FUNCTION_BLOCK FB_ComplexSheetStackerControl
VAR_INPUT

    //==============================================================
    // Group command inputs
    //==============================================================
    startCmd                            : BOOL;
    stopCmd                             : BOOL;
    resetCmd                            : BOOL;


    //==============================================================
    // Speed reference inputs
    //==============================================================
    lineSpeedMPM                        : REAL;

    // EN: Current sheet length [mm].
    // PT: Comprimento atual da chapa [mm].
    sheetLengthMm                       : REAL;


    //==============================================================
    // Package command input
    //==============================================================
    // EN: Rising edge starts package separation cycle.
    // PT: Borda de subida inicia o ciclo de separação do pacote.
    packageCompleteCmd                  : BOOL;
	sheetConveyorsSpeedUpCmd : BOOL;

    //==============================================================
    // Machine configuration
    //==============================================================
    machineConfig                       : ComplexStackerConfig_TypeStruct;


    //==============================================================
    // Safety input
    //==============================================================
    safetyCircuitOk                     : BOOL;


    //==============================================================
    // Synchronized conveyor drive status inputs
    //==============================================================
    sheetConveyor1DriveOk               : BOOL;
    sheetConveyor2DriveOk               : BOOL;
    sheetConveyor3DriveOk               : BOOL;
    sheetConveyor4DriveOk               : BOOL;
    elevatorDriveOk              : BOOL;


    //==============================================================
    // Auxiliary drive status inputs
    //==============================================================
    backstopDriveOk                     : BOOL;

	//==============================================================
	// Sheet stack discharge conveyor drive status input
	//==============================================================
    sheetStackDischargeConveyorDriveOk                 : BOOL;

	//==============================================================
	// EN: Stack buffer conveyor drive status inputs
	// PT: Entradas de estado dos acionamentos das esteiras buffer
	//==============================================================
	stackBufferConveyor1DriveOk            : BOOL;
	stackBufferConveyor2DriveOk            : BOOL;
	stackBufferConveyor3DriveOk            : BOOL;

	//==============================================================
	// EN: Stack detection sensors
	// PT: Sensores de detecção das pilhas
	//==============================================================
	stackBufferConveyor1StackPresentSensor : BOOL;
	stackBufferConveyor2StackPresentSensor : BOOL;
	stackBufferConveyor3StackPresentSensor : BOOL;
	elevatorStackPresentSensor             : BOOL;
	elevatorStackExitClearSensor           : BOOL;
	backstopMaterialInterlockSensor         : BOOL;
	backstopStackLevelSensor                : BOOL;

	
    //==============================================================
    // Position / measurement inputs
    //==============================================================
    stackHeightMm                       : REAL;
    backstopPositionMm                  : REAL;
    elevatorPositionMm           : REAL;


	//==============================================================
	// Elevator command inputs
	//==============================================================
	// EN: Starts elevator homing cycle.
	// PT: Inicia o ciclo de homing do elevador.
	elevatorHomeCmd              : BOOL;
	
	// EN: Enables elevator automatic mode. Auto-home is requested on
	//     startCmd and automatic leveling uses the stack level sensor.
	// PT: Habilita o modo automático do elevador. O auto-home é solicitado
	//     no startCmd e o nivelamento automático usa o sensor de nível da pilha.
	elevatorAutoCmd              : BOOL;
	
	// EN: Jog-up command in manual mode or during automatic leveling.
	// PT: Comando de jog para subir no manual ou durante o nivelamento automático.
	elevatorUpCmd                : BOOL;
	
	// EN: Jog-down command in manual mode or during automatic leveling.
	// PT: Comando de jog para descer no manual ou durante o nivelamento automático.
	elevatorDownCmd              : BOOL;


    //==============================================================
    // Elevator limit inputs
    //==============================================================
    elevatorUpperSafetyLimit     : BOOL;
    elevatorLowerSafetyLimit     : BOOL;

    elevatorUpperLimit           : BOOL;
    elevatorLowerLimit           : BOOL;


    //==============================================================
    // Backstop command inputs
    //==============================================================
    // EN: Starts the backstop homing cycle.
    // PT: Inicia o ciclo de homing do backstop.
    backstopHomeCmd                     : BOOL;
	
    // EN: Starts the backstop homing cycle.
    // PT: Inicia o ciclo de homing do backstop.
    backstopExecutePositioningCmd			 : BOOL;
    // EN: Enables automatic positioning according to sheet length.
    // PT: Habilita posicionamento automático conforme comprimento da chapa.
    backstopAutoCmd                     : BOOL;

    // EN: Manual open command.
    // PT: Comando manual para abrir.
    backstopOpenCmd                     : BOOL;

    // EN: Manual close command.
    // PT: Comando manual para fechar.
    backstopCloseCmd                    : BOOL;


    //==============================================================
    // Backstop limit inputs
    //==============================================================
    backstopSafeMaxLimit                    : BOOL;	
    backstopMaxLimit                 	   	: BOOL;
    backstopMinLimit                   		: BOOL;
    backstopSafeMinLimit                    : BOOL;


    //==============================================================
    // Sheet handling command inputs
    //==============================================================
	sheetStackDischargeConveyorManualRunCmd : BOOL;
    noCrushRollersDownCmd                 	: BOOL;

	// EN: Runs all three stack buffer conveyors.
	// PT: Aciona as três esteiras buffer de pilhas.
	stackBufferConveyorsRunCmd               : BOOL;

END_VAR


VAR_OUTPUT

	hmiAlarms : hmiAlarmsComplexStacker_TypeStruct;
	hmiStatus : hmiStatusComplexStacker_TypeStruct;
	stackerRunning : BOOL;
	alarmActive	: BOOL;
	stopMachinePulse : BOOL;
	reset 	: BOOL;
    //==============================================================
    // Synchronized conveyor drive outputs
    //==============================================================
    sheetConveyor1Run                   : BOOL;
    sheetConveyor2Run                   : BOOL;
    sheetConveyor3Run                   : BOOL;
    sheetConveyor4Run                   : BOOL;
	
	//==============================================================
	// Elevator drive outputs
	//==============================================================
	// EN: Elevator up run command.
	// PT: Comando para subir o elevador.
	elevatorRunUp                : BOOL;
	
	// EN: Elevator down run command.
	// PT: Comando para descer o elevador.
	elevatorRunDown              : BOOL;
	
	//==============================================================
	// Elevator magnetic brake output
	//==============================================================
	// EN: Magnetic brake release output. TRUE = brake released.
	// PT: Saída de liberação do freio magnético. TRUE = freio liberado.
	elevatorBrakeRelease         : BOOL;	

	// EN: Enables the elevator servo together with the stacker control.
	//     The servo remains enabled while stopped with zero speed reference.
	// PT: Habilita o servo do elevador junto com o controle do stacker.
	//     O servo permanece habilitado quando parado com referência zero.
	elevatorDriveEnable          : BOOL;

    //==============================================================
    // Backstop drive outputs
    //==============================================================
    // EN: Backstop forward run command. Positive/opening direction.
    // PT: Comando frente do backstop. Direção positiva/abrir.
    backstopRunFw                       : BOOL;

    // EN: Backstop reverse run command. Negative/closing direction.
    // PT: Comando reverso do backstop. Direção negativa/fechar.
    backstopRunRev                      : BOOL;

    // EN: Enables the backstop servo together with the stacker control.
    // PT: Habilita o servo do backstop junto com o controle do stacker.
    backstopDriveEnable                 : BOOL;

	//==============================================================
	// Sheet stack discharge conveyor outputs
	//==============================================================
	// EN: Sheet stack discharge conveyor run command.
	// PT: Comando de giro da esteira de descarga da pilha.
	sheetStackDischargeConveyorRun          : BOOL;

	//==============================================================
	// EN: Stack buffer conveyor run outputs
	// PT: Saídas de acionamento das esteiras buffer de pilhas
	//==============================================================
	stackBufferConveyor1Run                 : BOOL;
	stackBufferConveyor2Run                 : BOOL;
	stackBufferConveyor3Run                 : BOOL;




    //==============================================================
    // Synchronized conveyor speed reference outputs
    //==============================================================
    sheetConveyor1SpeedRefMPM           : REAL;
    sheetConveyor2SpeedRefMPM           : REAL;
    sheetConveyor3SpeedRefMPM           : REAL;
    sheetConveyor4SpeedRefMPM           : REAL;

    // EN: Signed elevator speed reference [mm/s]. Positive moves up
    //     and negative moves down.
    // PT: Referência de velocidade com sinal do elevador [mm/s].
    //     Positivo sobe e negativo desce.
    elevatorSpeedRefMmps                 : REAL;
	// EN: Sheet stack discharge conveyor speed reference [m/min].
	// PT: Referência de velocidade da esteira de descarga da pilha [m/min].
	sheetStackDischargeConveyorSpeedRefMPM  : REAL;

	// EN: Stack buffer conveyor speed references [m/min].
	// PT: Referências de velocidade das esteiras buffer [m/min].
	stackBufferConveyor1SpeedRefMPM         : REAL;
	stackBufferConveyor2SpeedRefMPM         : REAL;
	stackBufferConveyor3SpeedRefMPM         : REAL;

	// EN: TRUE while all three stack buffer positions are occupied.
	// PT: TRUE enquanto as três posições buffer estiverem ocupadas.
	stackBufferFull                         : BOOL;

	// EN: Requests the parent controller to reduce the machine speed.
	// PT: Solicita ao controlador pai a redução da velocidade da máquina.
	lineSpeedReductionRequest               : BOOL;

    //==============================================================
    // Backstop speed reference output
    //==============================================================
    // EN: Signed backstop speed reference [mm/s]. Positive opens and negative closes.
    // PT: Referência de velocidade com sinal do backstop [mm/s]. Positivo abre e negativo fecha.
    backstopSpeedRefMmps                : REAL;
	
	
	
    backstopPlateUpSolenoid                : BOOL;


    //==============================================================
    // Backstop encoder set outputs
    //==============================================================
    // EN: Pulse output to set/reset backstop encoder position.
    // PT: Pulso de saída para setar/resetar a posição do encoder do backstop.
    backstopSetEncoderPosition          : BOOL;

    // EN: Position value to set in the encoder block [mm].
    // PT: Valor de posição a ser gravado no bloco do encoder [mm].
    backstopSetEncoderPositionMm        : REAL;


    //==============================================================
    // Pneumatic valve outputs
    //==============================================================
    brakeValve                          : BOOL;

    sheetBrush1Valve                    : BOOL;
    sheetBrush2Valve                    : BOOL;
    sheetBrush3Valve                    : BOOL;

    brakeBrushValve                     : BOOL;
    backstopUpValve                     : BOOL;
    noCrushRollersUpDownValve               : BOOL;


    //==============================================================
    // General status outputs
    //==============================================================
    deviceState                         : STRING(30);

    faultActive                         : BOOL;
    synchronizedConveyorsRunning        : BOOL;


    //==============================================================
    // Sheet stack separation status outputs
    //==============================================================
    sheetStackSeparationState           : STRING(30);
    sheetStackSeparationStateCode       : INT;

    sheetStackSeparationReady           : BOOL;
    sheetStackSeparationActive          : BOOL;

    // EN: One-scan pulse when sheet stack separation starts.
    // PT: Pulso de um ciclo quando inicia a separação da pilha de chapas.
    sheetStackSeparationStarted         : BOOL;

    // EN: One-scan pulse when sheet stack separation finishes.
    // PT: Pulso de um ciclo quando finaliza a separação da pilha de chapas.
    sheetStackSeparationFinished        : BOOL;

    // EN: Brake active during sheet stack separation.
    // PT: Freio ativo durante a separação da pilha de chapas.
    sheetStackBrakeActive               : BOOL;


    //==============================================================
    // Sheet conveyor 2 separation status outputs
    //==============================================================
    sheetConveyor2SeparationActive      : BOOL;

    // EN: One-scan pulse when conveyor 2 separation tracking starts.
    // PT: Pulso de um ciclo quando inicia o rastreamento de separação da esteira 2.
    sheetConveyor2SeparationStarted     : BOOL;

    // EN: One-scan pulse when conveyor 2 separation tracking finishes.
    // PT: Pulso de um ciclo quando finaliza o rastreamento de separação da esteira 2.
    sheetConveyor2SeparationFinished    : BOOL;

    sheetConveyor2HighSpeedActive       : BOOL;

    // EN: Current conveyor 2 separation tracking distance [m].
    // PT: Distância atual rastreada na separação da esteira 2 [m].
    sheetConveyor2TrackingDistanceM     : REAL;

    // EN: Conveyor 2 separation target distance [m].
    // PT: Distância alvo de separação da esteira 2 [m].
    sheetConveyor2TargetDistanceM       : REAL;


    //==============================================================
    // Sheet conveyor 3 separation status outputs
    //==============================================================
    sheetConveyor3SeparationActive      : BOOL;

    // EN: One-scan pulse when conveyor 3 separation tracking starts.
    // PT: Pulso de um ciclo quando inicia o rastreamento de separação da esteira 3.
    sheetConveyor3SeparationStarted     : BOOL;

    // EN: One-scan pulse when conveyor 3 separation tracking finishes.
    // PT: Pulso de um ciclo quando finaliza o rastreamento de separação da esteira 3.
    sheetConveyor3SeparationFinished    : BOOL;

    sheetConveyor3HighSpeedActive       : BOOL;

    // EN: Current conveyor 3 separation tracking distance [m].
    // PT: Distância atual rastreada na separação da esteira 3 [m].
    sheetConveyor3TrackingDistanceM     : REAL;

    // EN: Conveyor 3 separation target distance [m].
    // PT: Distância alvo de separação da esteira 3 [m].
    sheetConveyor3TargetDistanceM       : REAL;

    //==============================================================
    // Sheet conveyor 4 separation status outputs
    //==============================================================
    sheetConveyor4SeparationActive      : BOOL;
    sheetConveyor4SeparationStarted     : BOOL;
    sheetConveyor4SeparationFinished    : BOOL;
    sheetConveyor4HighSpeedActive       : BOOL;
    sheetConveyor4TrackingDistanceM     : REAL;
    sheetConveyor4TargetDistanceM       : REAL;

	//==============================================================
	// Elevator encoder set outputs
	//==============================================================
	// EN: Pulse output to set/reset elevator encoder position.
	// PT: Pulso de saída para setar/resetar a posição do encoder do elevador.
	elevatorSetEncoderPosition   : BOOL;
	
	// EN: Position value to set in the elevator encoder block [mm].
	// PT: Valor de posição a ser gravado no bloco do encoder do elevador [mm].
	elevatorSetEncoderPositionMm : REAL;
	
	
	//==============================================================
	// Elevator status outputs
	//==============================================================
	elevatorState                : STRING(30);
	
	elevatorHomed                : BOOL;
	elevatorInPosition           : BOOL;

	// EN: TRUE when the homed elevator is at or below the configured
	//     minimum position considering the position tolerance.
	// PT: TRUE quando o elevador referenciado está na posição mínima
	//     configurada ou abaixo dela, considerando a tolerância.
	elevatorAtMinPosition        : BOOL;

	// EN: TRUE when the homed elevator is at or above the configured
	//     maximum position considering the position tolerance.
	// PT: TRUE quando o elevador referenciado está na posição máxima
	//     configurada ou acima dela, considerando a tolerância.
	elevatorAtMaxPosition        : BOOL;

	// EN: TRUE while manual jog speed is reduced near the endpoint
	//     toward which the elevator is moving.
	// PT: TRUE enquanto a velocidade do jog manual estiver reduzida próximo
	//     da extremidade para a qual o elevador está se movimentando.
	elevatorManualLowSpeedZoneActive : BOOL;

	elevatorFault                : BOOL;
	elevatorFaultCode            : INT;
	
	// EN: Current calculated elevator target position [mm].
	// PT: Posição alvo calculada atual do elevador [mm].
	elevatorTargetPositionMm     : REAL;
	
	// EN: Current elevator position error [mm].
	// PT: Erro atual de posição do elevador [mm].
	elevatorPositionErrorMm      : REAL;

    //==============================================================
    // Backstop status outputs
    //==============================================================
    backstopState                       : STRING(30);

    backstopHomed                       : BOOL;
    backstopInPosition                  : BOOL;
    backstopFault                       : BOOL;
    backstopFaultCode                   : INT;

    // EN: Current calculated target position [mm].
    // PT: Posição alvo calculada atualmente [mm].
    backstopTargetPositionMm            : REAL;

    // EN: Current position error [mm].
    // PT: Erro atual de posição [mm].
    backstopPositionErrorMm             : REAL;
	
	//==============================================================
	// Sheet stack discharge conveyor control state
	//==============================================================
	sheetStackDischargeConveyorState               : STRING(30);
	sheetStackDischargeConveyorFault               : BOOL;
	sheetStackDischargeConveyorFaultCode           : INT;
	
	//==============================================================
	// Sheet stack discharge sequence status outputs
	//==============================================================
	sheetStackDischargeState                : STRING(30);
	sheetStackDischargeStateCode            : INT;
	
	sheetStackDischargePending              : BOOL;
	sheetStackDischargeActive               : BOOL;
	sheetStackDischargeStarted              : BOOL;
	sheetStackDischargeFinished             : BOOL;
	
	sheetStackDischargeFault                : BOOL;
	sheetStackDischargeFaultCode            : INT;
	
	//==============================================================
	// Sheet stack discharge last cycle diagnostic outputs
	//==============================================================
	sheetStackDischargeLastCycleOk          : BOOL;
	sheetStackDischargeLastResultCode       : INT;
	sheetStackDischargeLastFaultStepCode    : INT;
	sheetStackDischargeLastFaultCode        : INT;	

END_VAR

VAR
	
	//==============================================================
	// Stop machine pulse control
	//==============================================================
	stopMachineFaultCondition     : BOOL;
	stopMachineFaultConditionOld  : BOOL;
	rStopMachineFaultCondition    : BOOL;
	
	tpStopMachinePulse            : TP;
	
	//==============================================================
	// Backstop manual intervention memory
	//==============================================================
	backstopManualInterventionActive     : BOOL;
	backstopManualInterventionPositionMm : REAL;
	
	//==============================================================
	// Sheet stack discharge backstop latched targets
	//==============================================================
	backstopProgrammedDischargeTargetMm : REAL;
	backstopDischargeOpenBasePositionMm : REAL;
	backstopDischargeOpenTargetMm       : REAL;
	
	//==============================================================
	// Backstop automatic positioning command control
	//==============================================================
	backstopExecutePositioningCmdOld    : BOOL;
	rBackstopExecutePositioning         : BOOL;
	
	backstopTargetOverrideOld           : BOOL;
	backstopTargetOverrideFallingEdge   : BOOL;
	
	backstopPositioningRequestActive    : BOOL;
	backstopLatchedTargetPositionMm     : REAL;
	backstopProgrammedTargetPositionMm  : REAL;
	
	//==============================================================
	// Backstop manual intervention memory
	//==============================================================
	// EN: Used by automatic discharge sequence to avoid closing onto material
	//     after operator manual intervention.

	//==============================================================
	// Backstop encoder set pulse
	//==============================================================
	backstopSetEncoderPositionTrigger  : BOOL;
	tpBackstopSetEncoderPosition       : TP;

	//==============================================================
	// Sheet stack discharge backstop latched targets
	//==============================================================

    //==============================================================
    // Group state machine
    //==============================================================
    syncConveyorsState                  : INT;


    //==============================================================
    // Package separation state machine
    //==============================================================
    packageSeparationState              : INT;


    //==============================================================
    // Backstop state machine
    //==============================================================
    backstopControlState                : INT;


    //==============================================================
    // Edge detection
    //==============================================================
    startCmdOld                         : BOOL;
    stopCmdOld                          : BOOL;
    packageCompleteCmdOld               : BOOL;

    backstopHomeCmdOld                  : BOOL;


    //==============================================================
    // Internal conditions
    //==============================================================
    allSynchronizedDrivesOk             : BOOL;
    anyFault                            : BOOL;
    speedControlEnabled                 : BOOL;
    rampReset                           : BOOL;


    //==============================================================
    // Sheet length conversion
    //==============================================================
    // EN: Internal sheet length converted from mm to m.
    // PT: Comprimento interno da chapa convertido de mm para m.
    sheetLengthM                        : REAL;


    //==============================================================
    // Normal speed calculation
    //==============================================================
    normalStackerSpeedMPM               : REAL;

    sheetConveyor1NormalSpeedMPM        : REAL;
    sheetConveyor2NormalSpeedMPM        : REAL;
    sheetConveyor3NormalSpeedMPM        : REAL;
    sheetConveyor4NormalSpeedMPM        : REAL;
    elevatorNormalSpeedMPM       : REAL;


    //==============================================================
    // Package gap speed calculation
    //==============================================================
    sheetConveyor2GapSpeedMPM           : REAL;
    sheetConveyor3GapSpeedMPM           : REAL;
    sheetConveyor4GapSpeedMPM           : REAL;


    //==============================================================
    // Speed targets
    //==============================================================
    sheetConveyor1TargetSpeedMPM        : REAL;
    sheetConveyor2TargetSpeedMPM        : REAL;
    sheetConveyor3TargetSpeedMPM        : REAL;
    sheetConveyor4TargetSpeedMPM        : REAL;
    elevatorTargetSpeedMPM       : REAL;


    //==============================================================
    // Package gap distance calculation
    //==============================================================
    packageGapDistanceTargetM           : REAL;

    sheetConveyor2OpeningSpeedMPM       : REAL;
    sheetConveyor3OpeningSpeedMPM       : REAL;
    sheetConveyor4OpeningSpeedMPM       : REAL;

    sheetConveyor2OpeningDistanceM      : REAL;
    sheetConveyor3OpeningDistanceM      : REAL;
    sheetConveyor4OpeningDistanceM      : REAL;


	//==============================================================
	// Elevator state machine
	//==============================================================
	elevatorControlState         : INT;
	
	
	//==============================================================
	// Elevator edge detection
	//==============================================================
	elevatorHomeCmdOld           : BOOL;
	rElevatorHome                : BOOL;
	
	
	//==============================================================
	// Elevator encoder set pulse
	//==============================================================
	elevatorSetEncoderPositionTrigger   : BOOL;
	tpElevatorSetEncoderPosition        : TP;
	
	
	//==============================================================
	// Elevator control calculation
	//==============================================================
	elevatorAutoTargetPositionMm        : REAL;
	elevatorRawSpeedRefMmps             : REAL;
	
	// EN: Internal signed speed command. Positive = up, negative = down.
	// PT: Comando interno de velocidade com sinal. Positivo = subir, negativo = descer.
	elevatorSignedSpeedRefMmps          : REAL;
	
	elevatorAbsPositionErrorMm          : REAL;
	
	
	//==============================================================
	// Elevator movement permissions
	//==============================================================
	elevatorUpAllowed                   : BOOL;
	elevatorDownAllowed                 : BOOL;
	
	elevatorMoveRequest                 : BOOL;
	elevatorBrakeReleaseRequest         : BOOL;
	
	
	//==============================================================
	// Elevator homing
	//==============================================================
	elevatorHomeLimitReached            : BOOL;
	elevatorHomeDownAllowed             : BOOL;
	elevatorHomeReleaseAllowed          : BOOL;
	elevatorManualCommandArmed          : BOOL;
	elevatorManualCommandRequest        : BOOL;
	elevatorReadyForAutomaticCycle      : BOOL;
	
	
	//==============================================================
	// Elevator timers
	//==============================================================
	tonElevatorHomingTimeout            : TON;
	tonElevatorHomeSettleDelay          : TON;
	tonElevatorLevelingSpeed2Delay      : TON;
	
	// EN: Delay after brake release before motor movement.
	// PT: Atraso após liberar o freio antes de movimentar o motor.
	tonElevatorBrakeReleaseDelay        : TON;
	
	// EN: Keeps brake released for a short time after movement stops.
	// PT: Mantém o freio liberado por um tempo após parar o movimento.
	tonElevatorBrakeHoldDelay           : TON;
	
	
	//==============================================================
	// Elevator speed ramp instance
	//==============================================================
	// EN: Ramp used for elevator vertical speed [mm/s].
	// PT: Rampa usada para velocidade vertical do elevador [mm/s].
	instRampElevator                    : FB_Gen_SRamp;
	

    //==============================================================
    // Backstop control calculation
    //==============================================================
    backstopAutoTargetPositionMm        : REAL;
    backstopRawSpeedRefMmps             : REAL;
    backstopAbsPositionErrorMm          : REAL;

    backstopHomeLimitReached            : BOOL;
    backstopOpenAllowed                 : BOOL;
    backstopCloseAllowed                : BOOL;

    rBackstopHome                       : BOOL;


	//==============================================================
	// Backstop homing edge detection
	//==============================================================
	backstopHomeLimitOld                 : BOOL;
	backstopHomeLimitFallingEdge         : BOOL;
	backstopHomeMoveAllowed              : BOOL;
	
	
	
	//==============================================================
	// Backstop timers
	//==============================================================
	tonBackstopHomeSettleDelay           : TON;



    //==============================================================
    // Backstop timers
    //==============================================================
    tonBackstopHomingTimeout            : TON;


    //==============================================================
    // Speed ramp instances
    //==============================================================
    instRampSheetConveyor1              : FB_Gen_SRamp;
    instRampSheetConveyor2              : FB_Gen_SRamp;
    instRampSheetConveyor3              : FB_Gen_SRamp;
    instRampSheetConveyor4              : FB_Gen_SRamp;


    //==============================================================
    // PLC scan time measurement
    //==============================================================
    instCycleTime                       : CYCLE_TIME;
    scanTimeS                           : REAL;
    scanTimeMs                          : REAL;

	backstopSignedSpeedRefMmps: REAL;
	
	//==============================================================
	// Sheet stack discharge state machine
	//==============================================================
	sheetStackDischargeControlState         : INT;
	
	
	//==============================================================
	// Sheet stack discharge edge detection
	//==============================================================
	packageCompleteCmdOldDischarge          : BOOL;
	rPackageCompleteDischarge               : BOOL;
	
	
	//==============================================================
	// Sheet stack discharge timers
	//==============================================================
	tonSheetStackDischarge                  : TON;
	tonSheetStackDischargePlatformClearTimeout : TON;
	elevatorPlatformClearDetected           : BOOL;
	elevatorStackPresentAtDischargeStart    : BOOL;
	
	
	//==============================================================
	// Sheet stack discharge internal conditions
	//==============================================================
	sheetStackDischargeFaultCondition       : BOOL;
	
	
	//==============================================================
	// Backstop target override
	//==============================================================
	backstopTargetOverrideActive            : BOOL;
	backstopTargetOverridePositionMm        : REAL;
	backstopRequiredForAutomaticOperation   : BOOL;
	
	
	//==============================================================
	// Elevator target override
	//==============================================================
	elevatorTargetOverrideActive     : BOOL;
	elevatorTargetOverridePositionMm : REAL;	
	
	
	sheetStackDischargeConveyorRunRequest: BOOL;
	instTONBackstopDownDelay: TON;
	
	//==============================================================
	// Sheet stack discharge step timeout
	//==============================================================
	tonSheetStackDischargeStepTimeout       : TON;
	
	sheetStackDischargeCycleHasManualSkip   : BOOL;
	sheetStackDischargeCycleHasTimeout      : BOOL;	
	
	
	//==============================================================
	// Elevator homing edge detection
	//==============================================================
	elevatorHomeLimitOld                 : BOOL;
	elevatorHomeLimitFallingEdge         : BOOL;	

	//==============================================================
	// System master run control
	//==============================================================
	systemRunEnable : BOOL;
	
	rStartCmd : BOOL;
	rStopCmd  : BOOL;
	
	//==============================================================
	// Automatic homing requests generated by master start
	//==============================================================
	backstopAutoHomeRequest        : BOOL;
	elevatorAutoHomeRequest : BOOL;
	
	//==============================================================
	// Elevator home request command control
	//==============================================================
	elevatorHomeRequestCombined    : BOOL;
	elevatorHomeRequestCombinedOld : BOOL;
	backstopHomeRunning: BOOL;
	//==============================================================
	// Backstop home request command control
	//==============================================================
	backstopHomeRequestCombined    : BOOL;
	backstopHomeRequestCombinedOld : BOOL;

	//==============================================================
	// EN: Stack buffer conveyor control
	// PT: Controle das esteiras buffer de pilhas
	//==============================================================
	stackBufferControlState                 : INT;
	stackBufferTargetConveyor               : INT;
	elevatorStackExitClearSensorOld         : BOOL;
	rElevatorStackExitClear                 : BOOL;
	tonStackBufferStopDelay                 : TON;
	tonStackBufferTransferTimeout           : TON;
	tonStackBufferFullSpeedReduction        : TON;
	
END_VAR

_SystemControl();

_SheetConveyorGroupControl();
_ConveyorSpeedControl();

_SheetStackDischargeControl();

_BackstopControl();
_ElevatorControl();
_SheetStackDischargeConveyorControl();
_StackBufferConveyorsControl();
_MachineAuxilary();
_HmiStatus();
_AlarmControl();

//==============================================================
// COMPLEX STACKER — ALARM CONTROL
// EN: Maps internal faults and status conditions to HMI alarm structure.
//==============================================================
METHOD _AlarmControl

VAR
	hmiAlarmsNotActive: hmiAlarmsComplexStacker_TypeStruct;
END_VAR
//==============================================================
// HMI alarms reset / latch logic
//==============================================================

IF resetCmd THEN

    // Reset geral dos alarmes
    hmiAlarms := hmiAlarmsNotActive;

ELSE

    //==============================================================
    // 1) General / system alarms
    //==============================================================
    hmiAlarms.safetyCircuitNotOk :=
        hmiAlarms.safetyCircuitNotOk OR
        NOT safetyCircuitOk;

    hmiAlarms.systemFaultActive :=
        hmiAlarms.systemFaultActive OR
        faultActive OR
        (
            backstopRequiredForAutomaticOperation AND
            backstopFault
        ) OR
        elevatorFault OR
        sheetStackDischargeFault OR
        sheetStackDischargeConveyorFault OR
        NOT stackBufferConveyor1DriveOk OR
        NOT stackBufferConveyor2DriveOk OR
        NOT stackBufferConveyor3DriveOk;

    hmiAlarms.systemNotEnabled :=
        hmiAlarms.systemNotEnabled OR
        NOT systemRunEnable;


    //==============================================================
    // 2) Sheet conveyor group alarms
    //==============================================================
    hmiAlarms.sheetConveyor1DriveNotOk :=
        hmiAlarms.sheetConveyor1DriveNotOk OR
        NOT sheetConveyor1DriveOk;

    hmiAlarms.sheetConveyor2DriveNotOk :=
        hmiAlarms.sheetConveyor2DriveNotOk OR
        NOT sheetConveyor2DriveOk;

    hmiAlarms.sheetConveyor3DriveNotOk :=
        hmiAlarms.sheetConveyor3DriveNotOk OR
        NOT sheetConveyor3DriveOk;

    hmiAlarms.sheetConveyor4DriveNotOk :=
        hmiAlarms.sheetConveyor4DriveNotOk OR
        NOT sheetConveyor4DriveOk;

    hmiAlarms.sheetConveyorGroupFault :=
        hmiAlarms.sheetConveyorGroupFault OR
        NOT safetyCircuitOk OR
        NOT sheetConveyor1DriveOk OR
        NOT sheetConveyor2DriveOk OR
        NOT sheetConveyor3DriveOk OR
        NOT sheetConveyor4DriveOk;


    //==============================================================
    // 2.1) Stack buffer conveyor alarms
    // EN: Buffer drive faults are alarmed without stopping the main
    //     synchronized conveyor group automatically.
    // PT: Falhas dos drives do buffer geram alarme sem parar automaticamente
    //     o grupo principal de esteiras sincronizadas.
    //==============================================================
    hmiAlarms.stackBufferConveyor1DriveNotOk :=
        hmiAlarms.stackBufferConveyor1DriveNotOk OR
        NOT stackBufferConveyor1DriveOk;

    hmiAlarms.stackBufferConveyor2DriveNotOk :=
        hmiAlarms.stackBufferConveyor2DriveNotOk OR
        NOT stackBufferConveyor2DriveOk;

    hmiAlarms.stackBufferConveyor3DriveNotOk :=
        hmiAlarms.stackBufferConveyor3DriveNotOk OR
        NOT stackBufferConveyor3DriveOk;

    hmiAlarms.stackBufferConveyorGroupFault :=
        hmiAlarms.stackBufferConveyorGroupFault OR
        NOT safetyCircuitOk OR
        NOT stackBufferConveyor1DriveOk OR
        NOT stackBufferConveyor2DriveOk OR
        NOT stackBufferConveyor3DriveOk;

 //   hmiAlarms.synchronizedConveyorsNotRunning :=
 //       hmiAlarms.synchronizedConveyorsNotRunning OR
 //       (
 //           systemRunEnable AND
 //           NOT synchronizedConveyorsRunning
 //       );


    //==============================================================
    // 3) Sheet stack separation alarms / indications
    //==============================================================
    // Mantido comentado conforme lógica original.
    // Se quiser ativar como latch, use o mesmo padrão:
    //
    // hmiAlarms.sheetStackSeparationNotReady :=
    //     hmiAlarms.sheetStackSeparationNotReady OR
    //     (
    //         systemRunEnable AND
    //         synchronizedConveyorsRunning AND
    //         NOT sheetStackSeparationReady
    //     );
    //
    // hmiAlarms.sheetStackSeparationActive :=
    //     hmiAlarms.sheetStackSeparationActive OR
    //     sheetStackSeparationActive;
    //
    // hmiAlarms.sheetStackBrakeActive :=
    //     hmiAlarms.sheetStackBrakeActive OR
    //     sheetStackBrakeActive;


    //==============================================================
    // 4) Sheet stack discharge sequence alarms / indications
    //==============================================================
    hmiAlarms.sheetStackDischargeFault :=
        hmiAlarms.sheetStackDischargeFault OR
        sheetStackDischargeFault;

    hmiAlarms.sheetStackDischargeLastCycleNotOk :=
        hmiAlarms.sheetStackDischargeLastCycleNotOk OR
        (
            NOT sheetStackDischargeLastCycleOk AND
            sheetStackDischargeLastResultCode <> 0
        );

    hmiAlarms.sheetStackDischargeTimeout :=
        hmiAlarms.sheetStackDischargeTimeout OR
        sheetStackDischargeLastResultCode = 3;

    hmiAlarms.sheetStackDischargeManualSkip :=
        hmiAlarms.sheetStackDischargeManualSkip OR
        sheetStackDischargeLastResultCode = 2;


    //==============================================================
    // 5) Sheet stack discharge conveyor alarms
    //==============================================================
    hmiAlarms.sheetStackDischargeConveyorDriveNotOk :=
        hmiAlarms.sheetStackDischargeConveyorDriveNotOk OR
        NOT sheetStackDischargeConveyorDriveOk;

    hmiAlarms.sheetStackDischargeConveyorFault :=
        hmiAlarms.sheetStackDischargeConveyorFault OR
        sheetStackDischargeConveyorFault;


    //==============================================================
    // 6) Backstop alarms / indications
    //==============================================================
    hmiAlarms.backstopDriveNotOk :=
        hmiAlarms.backstopDriveNotOk OR
        NOT backstopDriveOk;

    hmiAlarms.backstopFault :=
        hmiAlarms.backstopFault OR
        backstopFault;

    hmiAlarms.backstopNotHomed :=
        hmiAlarms.backstopNotHomed OR
        (
            backstopAutoCmd AND
            NOT backstopHomed
        );

    (*
    hmiAlarms.backstopNotInPosition :=
        hmiAlarms.backstopNotInPosition OR
        (
            systemRunEnable AND
            backstopAutoCmd AND
            backstopHomed AND
            NOT backstopInPosition AND
            NOT backstopTargetOverrideActive
        );
    *)

    hmiAlarms.backstopSafeMaxLimitActive :=
        hmiAlarms.backstopSafeMaxLimitActive OR
        backstopSafeMaxLimit;

    hmiAlarms.backstopSafeMinLimitActive :=
        hmiAlarms.backstopSafeMinLimitActive OR
        backstopSafeMinLimit;

    (*
    hmiAlarms.backstopMaxLimitActive :=
        hmiAlarms.backstopMaxLimitActive OR
        backstopMaxLimit;

    hmiAlarms.backstopMinLimitActive :=
        hmiAlarms.backstopMinLimitActive OR
        backstopMinLimit;

    hmiAlarms.backstopManualInterventionActive :=
        hmiAlarms.backstopManualInterventionActive OR
        backstopManualInterventionActive;
    *)


    //==============================================================
    // 7) Elevator alarms / indications
    //==============================================================
    hmiAlarms.elevatorDriveNotOk :=
        hmiAlarms.elevatorDriveNotOk OR
        NOT elevatorDriveOk;

    hmiAlarms.elevatorFault :=
        hmiAlarms.elevatorFault OR
        elevatorFault;

    hmiAlarms.elevatorNotHomed :=
        hmiAlarms.elevatorNotHomed OR
        (
            elevatorAutoCmd AND
            NOT elevatorHomed
        );

//    hmiAlarms.elevatorNotInPosition :=
//        hmiAlarms.elevatorNotInPosition OR
//        (
//            systemRunEnable AND
//            elevatorAutoCmd AND
//            elevatorHomed AND
//            NOT elevatorInPosition
//        );

    hmiAlarms.elevatorUpperSafetyLimitActive :=
        hmiAlarms.elevatorUpperSafetyLimitActive OR
        elevatorUpperSafetyLimit;

    hmiAlarms.elevatorLowerSafetyLimitActive :=
        hmiAlarms.elevatorLowerSafetyLimitActive OR
        elevatorLowerSafetyLimit;

    (*
    hmiAlarms.elevatorUpperLimitActive :=
        hmiAlarms.elevatorUpperLimitActive OR
        elevatorUpperLimit;

    hmiAlarms.elevatorLowerLimitActive :=
        hmiAlarms.elevatorLowerLimitActive OR
        elevatorLowerLimit;
    *)

END_IF;
END_METHOD

//==============================================================
// COMPLEX STACKER — BACKSTOP CONTROL
// EN: Controls the backstop axis with homing, manual movement,
//     automatic positioning, override positioning and protections.
//
// Signed speed convention:
// Positive = open
// Negative = close
//
// State code:
// 0  = STOP
// 10 = HOME_FAST_SEARCH
// 11 = HOME_SLOW_EXIT_SENSOR
// 12 = HOME_SET_ENCODER
// 13 = HOME_WAIT_AFTER_SET
// 14 = HOME_MOVE_TO_TARGET
// 20 = MANUAL
// 30 = AUTO_POSITION
// 40 = FAULT
//==============================================================
METHOD _BackstopControl



//==============================================================
// 1) Default internal commands
//==============================================================
// EN: Internal signed speed is reset every scan and set by the active state.
//     Positive = open, negative = close.
backstopSignedSpeedRefMmps := 0.0;

// EN: Internal trigger for encoder set pulse.
backstopSetEncoderPositionTrigger := FALSE;


//==============================================================
// 2) Edge detection
//==============================================================
// EN: Home can be requested manually by HMI or automatically by _SystemControl.
//     Automatic home is accepted only when backstopAutoCmd is enabled.
//     Movement is allowed only when master system run is enabled.
backstopHomeRequestCombined :=
    systemRunEnable AND
    (
        backstopHomeCmd OR
        (
            backstopAutoCmd AND
            backstopAutoHomeRequest
        )
    );

rBackstopHome :=
    backstopHomeRequestCombined AND
    NOT backstopHomeRequestCombinedOld;

backstopHomeRequestCombinedOld :=
    backstopHomeRequestCombined;


// EN: Execute positioning command edge.
//     This command only generates movement when system is enabled and backstop auto is enabled.
rBackstopExecutePositioning :=
    systemRunEnable AND
    backstopExecutePositioningCmd AND
    NOT backstopExecutePositioningCmdOld;

backstopExecutePositioningCmdOld := backstopExecutePositioningCmd;


// EN: Override falling edge.
//     Used as fallback to return to programmed position if override is released.
backstopTargetOverrideFallingEdge :=
    backstopTargetOverrideOld AND NOT backstopTargetOverrideActive;

backstopTargetOverrideOld := backstopTargetOverrideActive;


//==============================================================
// 3) Home limit selection and edge detection
//==============================================================
// EN: Home limit depends on configured homing direction.
IF machineConfig.backstopHomeDirection > 0 THEN

    backstopHomeLimitReached := backstopMaxLimit;

ELSIF machineConfig.backstopHomeDirection < 0 THEN

    backstopHomeLimitReached := backstopMinLimit;

ELSE

    backstopHomeLimitReached := FALSE;

END_IF;


// EN: Falling edge is used after the home limit has been reached.
backstopHomeLimitFallingEdge :=
    backstopHomeLimitOld AND NOT backstopHomeLimitReached;

backstopHomeLimitOld := backstopHomeLimitReached;


//==============================================================
// 4) Movement permissions
//==============================================================
backstopOpenAllowed :=
    systemRunEnable AND
    safetyCircuitOk AND
    backstopDriveOk AND
    NOT backstopMaxLimit AND
    NOT backstopSafeMaxLimit AND
    (
        (NOT backstopHomed) OR
        (backstopPositionMm < machineConfig.backstopMaxPositionMm)
    );

backstopCloseAllowed :=
    systemRunEnable AND
    safetyCircuitOk AND
    backstopDriveOk AND
    NOT backstopMinLimit AND
    NOT backstopSafeMinLimit AND
    (
        (NOT backstopHomed) OR
        (backstopPositionMm > machineConfig.backstopMinPositionMm)
    );


// EN: During homing, the normal home limit is allowed.
//     Only the safe limit blocks movement.
IF machineConfig.backstopHomeDirection > 0 THEN

    backstopHomeMoveAllowed :=
        systemRunEnable AND
        safetyCircuitOk AND
        backstopDriveOk AND
        NOT backstopSafeMaxLimit;

ELSIF machineConfig.backstopHomeDirection < 0 THEN

    backstopHomeMoveAllowed :=
        systemRunEnable AND
        safetyCircuitOk AND
        backstopDriveOk AND
        NOT backstopSafeMinLimit;

ELSE

    backstopHomeMoveAllowed := FALSE;

END_IF;


//==============================================================
// 5) Programmed / override target calculation
//==============================================================
// EN: Programmed target follows sheet length plus mechanical offset.
//     This value can change, but it does not move the backstop by itself.
backstopProgrammedTargetPositionMm :=
    LIMIT(
        machineConfig.backstopMinPositionMm,
        MAX(0.0, sheetLengthMm) + machineConfig.backstopSheetLengthOffsetMm,
        machineConfig.backstopMaxPositionMm
    );


// EN: Before homing, keep the latched target updated with programmed target.
//     This avoids an invalid old target after power-up.
IF NOT backstopHomed THEN

    backstopLatchedTargetPositionMm := backstopProgrammedTargetPositionMm;

END_IF;


//==============================================================
// 5.1) Automatic positioning request handling
//==============================================================
// EN: Auto mode only enables positioning. It does not execute positioning.
//     Normal positioning must be requested by backstopExecutePositioningCmd.
//     Override positioning is requested by the automatic cycle.
IF NOT systemRunEnable THEN

    backstopPositioningRequestActive := FALSE;


ELSIF NOT backstopAutoCmd THEN

    backstopPositioningRequestActive := FALSE;


ELSIF backstopTargetOverrideActive THEN

    // EN: Override has priority. Clear normal positioning request.
    backstopPositioningRequestActive := FALSE;


ELSIF rBackstopExecutePositioning THEN

    // EN: Latch current programmed target only when execute command is received.
    backstopLatchedTargetPositionMm := backstopProgrammedTargetPositionMm;
    backstopPositioningRequestActive := TRUE;


ELSIF backstopTargetOverrideFallingEdge THEN

    // EN: Fallback after override release.
    //     The discharge sequence should normally keep override active
    //     during return. If override is released unexpectedly, return to
    //     programmed position automatically.
    backstopLatchedTargetPositionMm := backstopProgrammedTargetPositionMm;
    backstopPositioningRequestActive := TRUE;

END_IF;


//==============================================================
// 5.2) Active target selection
//==============================================================
// EN: Discharge override is accepted only while the backstop is in automatic.
//     In manual mode the backstop is completely independent from the cycle.
// PT: O override de descarte é aceito somente com o backstop em automático.
//     No modo manual o backstop fica completamente independente do ciclo.
IF systemRunEnable AND
   backstopAutoCmd AND
   backstopTargetOverrideActive THEN

    backstopTargetPositionMm :=
        LIMIT(
            machineConfig.backstopMinPositionMm,
            backstopTargetOverridePositionMm,
            machineConfig.backstopMaxPositionMm
        );

ELSE

    backstopTargetPositionMm :=
        LIMIT(
            machineConfig.backstopMinPositionMm,
            backstopLatchedTargetPositionMm,
            machineConfig.backstopMaxPositionMm
        );

END_IF;


//==============================================================
// 5.4) Home running flag
//==============================================================
IF (backstopControlState = 10) OR
   (backstopControlState = 11) OR
   (backstopControlState = 12) OR
   (backstopControlState = 13) OR
   (backstopControlState = 14) THEN

    backstopHomeRunning := TRUE;

ELSE

    backstopHomeRunning := FALSE;

END_IF;


//==============================================================
// 6) Position error calculation
//==============================================================
backstopPositionErrorMm :=
    backstopTargetPositionMm - backstopPositionMm;

backstopAbsPositionErrorMm :=
    ABS(backstopPositionErrorMm);

backstopInPosition :=
    backstopHomed AND
    (backstopAbsPositionErrorMm <= machineConfig.backstopPositionToleranceMm);


//==============================================================
// 7) Reset fault command
//==============================================================
IF resetCmd THEN

    IF safetyCircuitOk AND
       backstopDriveOk AND
       NOT backstopSafeMaxLimit AND
       NOT backstopSafeMinLimit THEN

        backstopFault := FALSE;
        backstopFaultCode := 0;

        IF backstopControlState = 40 THEN
            backstopControlState := 0;
        END_IF

    END_IF

END_IF;


//==============================================================
// 8) General protection
//==============================================================
IF NOT safetyCircuitOk THEN

    backstopState := 'SAFETY_OFF';

    tonBackstopHomingTimeout(IN := FALSE);
    tonBackstopHomeSettleDelay(IN := FALSE);

    backstopFault := TRUE;
    backstopFaultCode := 2;
    backstopControlState := 40;


ELSIF NOT backstopDriveOk THEN

    backstopState := 'DRIVE_NOT_OK';

    tonBackstopHomingTimeout(IN := FALSE);
    tonBackstopHomeSettleDelay(IN := FALSE);

    backstopFault := TRUE;
    backstopFaultCode := 1;
    backstopControlState := 40;


ELSIF backstopSafeMaxLimit THEN

    backstopState := 'SAFE_MAX_LIMIT';

    tonBackstopHomingTimeout(IN := FALSE);
    tonBackstopHomeSettleDelay(IN := FALSE);

    backstopFault := TRUE;
    backstopFaultCode := 6;
    backstopControlState := 40;


ELSIF backstopSafeMinLimit THEN

    backstopState := 'SAFE_MIN_LIMIT';

    tonBackstopHomingTimeout(IN := FALSE);
    tonBackstopHomeSettleDelay(IN := FALSE);

    backstopFault := TRUE;
    backstopFaultCode := 7;
    backstopControlState := 40;


ELSIF machineConfig.backstopHomeDirection = 0 THEN

    backstopState := 'INVALID_HOME_DIR';

    tonBackstopHomingTimeout(IN := FALSE);
    tonBackstopHomeSettleDelay(IN := FALSE);

    backstopFault := TRUE;
    backstopFaultCode := 5;
    backstopControlState := 40;


ELSIF NOT systemRunEnable THEN

    // EN: Master stop disables movement without generating an axis fault.
    backstopState := 'SYSTEM_DISABLED';

    backstopSignedSpeedRefMmps := 0.0;

    tonBackstopHomingTimeout(IN := FALSE);
    tonBackstopHomeSettleDelay(IN := FALSE);

    backstopPositioningRequestActive := FALSE;

    IF backstopControlState <> 40 THEN
        backstopControlState := 0;
    END_IF


ELSE

    //==============================================================
    // 9) Mode selection
    //==============================================================
    // EN: Homing has priority over manual and automatic positioning.
    IF rBackstopHome AND NOT backstopFault THEN
        backstopControlState := 10;
    END_IF;


    //==============================================================
    // 10) Backstop state machine
    //==============================================================
    CASE backstopControlState OF

        0: // STOP
            backstopState := 'STOP';

            tonBackstopHomingTimeout(IN := FALSE);
            tonBackstopHomeSettleDelay(IN := FALSE);

            // EN: Manual is allowed even with auto enabled,
            //     but not during an automatic cycle override.
            IF (backstopOpenCmd OR backstopCloseCmd) AND
               NOT (
                   backstopAutoCmd AND
                   backstopTargetOverrideActive
               ) THEN

                backstopControlState := 20;


            ELSIF backstopAutoCmd AND
                  (
                      backstopTargetOverrideActive OR
                      backstopPositioningRequestActive
                  ) THEN

                backstopControlState := 30;

            END_IF


        10: // HOME_FAST_SEARCH
            backstopState := 'HOME_FAST';

            backstopHomed := FALSE;
            backstopInPosition := FALSE;

            tonBackstopHomeSettleDelay(IN := FALSE);

            tonBackstopHomingTimeout(
                IN := TRUE,
                PT := machineConfig.backstopHomingTimeout
            );

            IF tonBackstopHomingTimeout.Q THEN

                backstopSignedSpeedRefMmps := 0.0;

                tonBackstopHomingTimeout(IN := FALSE);

                backstopFault := TRUE;
                backstopFaultCode := 3;

                backstopState := 'HOME_TIMEOUT';
                backstopControlState := 40;


            ELSIF backstopHomeLimitReached THEN

                backstopSignedSpeedRefMmps := 0.0;

                backstopControlState := 11;


            ELSE

                IF backstopHomeMoveAllowed THEN

                    IF machineConfig.backstopHomeDirection > 0 THEN

                        backstopSignedSpeedRefMmps :=
                            ABS(machineConfig.backstopHomingSpeedMmps);

                    ELSE

                        backstopSignedSpeedRefMmps :=
                            -ABS(machineConfig.backstopHomingSpeedMmps);

                    END_IF

                ELSE

                    backstopSignedSpeedRefMmps := 0.0;

                END_IF

            END_IF


        11: // HOME_SLOW_EXIT_SENSOR
            backstopState := 'HOME_SLOW_EXIT';

            tonBackstopHomeSettleDelay(IN := FALSE);

            tonBackstopHomingTimeout(
                IN := TRUE,
                PT := machineConfig.backstopHomingTimeout
            );

            IF tonBackstopHomingTimeout.Q THEN

                backstopSignedSpeedRefMmps := 0.0;

                tonBackstopHomingTimeout(IN := FALSE);

                backstopFault := TRUE;
                backstopFaultCode := 3;

                backstopState := 'HOME_TIMEOUT';
                backstopControlState := 40;


            ELSIF backstopHomeLimitFallingEdge THEN

                backstopSignedSpeedRefMmps := 0.0;

                tonBackstopHomingTimeout(IN := FALSE);

                backstopControlState := 12;


            ELSE

                IF backstopHomeMoveAllowed THEN

                    IF machineConfig.backstopHomeDirection > 0 THEN

                        backstopSignedSpeedRefMmps :=
                            -ABS(machineConfig.backstopMinMoveSpeedMmps);

                    ELSE

                        backstopSignedSpeedRefMmps :=
                            ABS(machineConfig.backstopMinMoveSpeedMmps);

                    END_IF

                ELSE

                    backstopSignedSpeedRefMmps := 0.0;

                END_IF

            END_IF


        12: // HOME_SET_ENCODER
            backstopState := 'HOME_SET_ENCODER';

            backstopSignedSpeedRefMmps := 0.0;

            tonBackstopHomingTimeout(IN := FALSE);
            tonBackstopHomeSettleDelay(IN := FALSE);

            // EN: Set encoder to configured known home position.
            backstopSetEncoderPositionTrigger := TRUE;
            backstopSetEncoderPositionMm := machineConfig.backstopHomePositionMm;

            backstopHomed := TRUE;
            backstopFault := FALSE;
            backstopFaultCode := 0;

            // EN: After homing, latch current programmed target for home move.
            backstopLatchedTargetPositionMm := backstopProgrammedTargetPositionMm;
            backstopPositioningRequestActive := TRUE;

            // EN: Homing cancels previous manual intervention memory.
            backstopManualInterventionActive := FALSE;
            backstopManualInterventionPositionMm := 0.0;

            backstopControlState := 13;


        13: // HOME_WAIT_AFTER_SET
            backstopState := 'HOME_WAIT';

            backstopSignedSpeedRefMmps := 0.0;

            tonBackstopHomingTimeout(IN := FALSE);

            // EN: Fixed wait after encoder set.
            tonBackstopHomeSettleDelay(
                IN := TRUE,
                PT := T#5S
            );

            IF tonBackstopHomeSettleDelay.Q THEN

                tonBackstopHomeSettleDelay(IN := FALSE);

                backstopControlState := 14;

            END_IF


        14: // HOME_MOVE_TO_TARGET
            backstopState := 'HOME_TO_TARGET';

            tonBackstopHomingTimeout(IN := FALSE);
            tonBackstopHomeSettleDelay(IN := FALSE);

            // EN: Move to the latched programmed target after homing.
            IF backstopInPosition THEN

                backstopSignedSpeedRefMmps := 0.0;

                backstopPositioningRequestActive := FALSE;

                // EN: Home positioning completed, no manual intervention pending.
                backstopManualInterventionActive := FALSE;
                backstopManualInterventionPositionMm := 0.0;

                backstopControlState := 0;


            ELSE

                backstopRawSpeedRefMmps :=
                    backstopPositionErrorMm * machineConfig.backstopPositionKp;

                backstopRawSpeedRefMmps :=
                    LIMIT(
                        -ABS(machineConfig.backstopAutoMaxSpeedMmps),
                        backstopRawSpeedRefMmps,
                        ABS(machineConfig.backstopAutoMaxSpeedMmps)
                    );

                IF ABS(backstopRawSpeedRefMmps) <
                   ABS(machineConfig.backstopMinMoveSpeedMmps) THEN

                    IF backstopPositionErrorMm > 0.0 THEN

                        backstopRawSpeedRefMmps :=
                            ABS(machineConfig.backstopMinMoveSpeedMmps);

                    ELSE

                        backstopRawSpeedRefMmps :=
                            -ABS(machineConfig.backstopMinMoveSpeedMmps);

                    END_IF

                END_IF

                IF (backstopRawSpeedRefMmps > 0.0) AND backstopOpenAllowed THEN

                    backstopSignedSpeedRefMmps := backstopRawSpeedRefMmps;

                ELSIF (backstopRawSpeedRefMmps < 0.0) AND backstopCloseAllowed THEN

                    backstopSignedSpeedRefMmps := backstopRawSpeedRefMmps;

                ELSE

                    backstopSignedSpeedRefMmps := 0.0;

                END_IF

            END_IF


        20: // MANUAL
            backstopState := 'MANUAL';

            tonBackstopHomingTimeout(IN := FALSE);
            tonBackstopHomeSettleDelay(IN := FALSE);

            // EN: An automatic override cancels manual control only when
            //     the backstop itself is enabled in automatic mode.
            // PT: O override automático cancela o controle manual somente
            //     quando o próprio backstop está habilitado em automático.
            IF backstopAutoCmd AND
               backstopTargetOverrideActive THEN

                backstopSignedSpeedRefMmps := 0.0;
                backstopControlState := 30;


            ELSIF backstopOpenCmd AND backstopCloseCmd THEN

                backstopSignedSpeedRefMmps := 0.0;


            ELSIF backstopOpenCmd THEN

                IF backstopOpenAllowed THEN

                    backstopSignedSpeedRefMmps :=
                        ABS(machineConfig.backstopManualSpeedMmps);

                    // EN: Store last manual intervention position.
                    //     This is updated while the operator holds the manual command.
                    backstopManualInterventionActive := TRUE;
                    backstopManualInterventionPositionMm := backstopPositionMm;

                ELSE

                    backstopSignedSpeedRefMmps := 0.0;

                END_IF


            ELSIF backstopCloseCmd THEN

                IF backstopCloseAllowed THEN

                    backstopSignedSpeedRefMmps :=
                        -ABS(machineConfig.backstopManualSpeedMmps);

                    // EN: Store last manual intervention position.
                    //     Even if operator closes, the discharge sequence will use
                    //     MAX(programmed position, manual position), so it remains safe.
                    backstopManualInterventionActive := TRUE;
                    backstopManualInterventionPositionMm := backstopPositionMm;

                ELSE

                    backstopSignedSpeedRefMmps := 0.0;

                END_IF


            ELSE

                backstopSignedSpeedRefMmps := 0.0;

                // EN: After manual command release, do not automatically return
                //     to programmed position. Wait for execute positioning command.
                backstopPositioningRequestActive := FALSE;

                backstopControlState := 0;

            END_IF


        30: // AUTO_POSITION
            backstopState := 'AUTO_POSITION';

            tonBackstopHomingTimeout(IN := FALSE);
            tonBackstopHomeSettleDelay(IN := FALSE);

            // EN: Manual mode always cancels automatic positioning,
            //     regardless of any external override request.
            // PT: O modo manual sempre cancela o posicionamento automático,
            //     independentemente de qualquer pedido externo de override.
            IF NOT backstopAutoCmd THEN

                backstopSignedSpeedRefMmps := 0.0;
                backstopPositioningRequestActive := FALSE;
                backstopControlState := 0;


            ELSIF NOT backstopHomed THEN

                backstopSignedSpeedRefMmps := 0.0;
                backstopState := 'AUTO_NO_HOME';


            ELSIF (backstopOpenCmd OR backstopCloseCmd) AND
                  NOT backstopTargetOverrideActive THEN

                // EN: Manual has priority only outside automatic cycle override.
                backstopSignedSpeedRefMmps := 0.0;
                backstopPositioningRequestActive := FALSE;
                backstopControlState := 20;


            ELSIF NOT backstopTargetOverrideActive AND
                  NOT backstopPositioningRequestActive THEN

                // EN: Auto enabled but no positioning command active.
                backstopSignedSpeedRefMmps := 0.0;
                backstopControlState := 0;


            ELSIF backstopInPosition THEN

                backstopSignedSpeedRefMmps := 0.0;

                // EN: Normal positioning command ends when target is reached.
                //     Override remains controlled by the automatic cycle.
                IF NOT backstopTargetOverrideActive THEN

                    backstopPositioningRequestActive := FALSE;

                    // EN: If the backstop returned to programmed target,
                    //     clear previous manual intervention memory.
                    backstopManualInterventionActive := FALSE;
                    backstopManualInterventionPositionMm := 0.0;

                    backstopControlState := 0;

                END_IF


            ELSE

                backstopRawSpeedRefMmps :=
                    backstopPositionErrorMm * machineConfig.backstopPositionKp;

                backstopRawSpeedRefMmps :=
                    LIMIT(
                        -ABS(machineConfig.backstopAutoMaxSpeedMmps),
                        backstopRawSpeedRefMmps,
                        ABS(machineConfig.backstopAutoMaxSpeedMmps)
                    );

                IF ABS(backstopRawSpeedRefMmps) <
                   ABS(machineConfig.backstopMinMoveSpeedMmps) THEN

                    IF backstopPositionErrorMm > 0.0 THEN

                        backstopRawSpeedRefMmps :=
                            ABS(machineConfig.backstopMinMoveSpeedMmps);

                    ELSE

                        backstopRawSpeedRefMmps :=
                            -ABS(machineConfig.backstopMinMoveSpeedMmps);

                    END_IF

                END_IF

                IF (backstopRawSpeedRefMmps > 0.0) AND backstopOpenAllowed THEN

                    backstopSignedSpeedRefMmps := backstopRawSpeedRefMmps;

                ELSIF (backstopRawSpeedRefMmps < 0.0) AND backstopCloseAllowed THEN

                    backstopSignedSpeedRefMmps := backstopRawSpeedRefMmps;

                ELSE

                    backstopSignedSpeedRefMmps := 0.0;

                END_IF

            END_IF


        40: // FAULT
            backstopState := 'FAULT';

            backstopSignedSpeedRefMmps := 0.0;

            tonBackstopHomingTimeout(IN := FALSE);
            tonBackstopHomeSettleDelay(IN := FALSE);

            backstopPositioningRequestActive := FALSE;

            IF resetCmd AND
               safetyCircuitOk AND
               backstopDriveOk AND
               NOT backstopSafeMaxLimit AND
               NOT backstopSafeMinLimit THEN

                backstopFault := FALSE;
                backstopFaultCode := 0;
                backstopControlState := 0;

            END_IF


    ELSE

        backstopControlState := 0;

    END_CASE;

END_IF;


//==============================================================
// 11) Encoder set pulse
//==============================================================
// EN: Extend encoder set command to ensure the encoder block sees it.
tpBackstopSetEncoderPosition(
    IN := backstopSetEncoderPositionTrigger,
    PT := machineConfig.backstopSetEncoderPulseTime
);

backstopSetEncoderPosition := tpBackstopSetEncoderPosition.Q;


//==============================================================
// 12) Backstop drive direction and speed outputs
//==============================================================
// EN: Convert signed internal speed command into direction outputs
//     and positive speed reference.
IF systemRunEnable AND
   safetyCircuitOk AND
   backstopDriveOk AND
   NOT backstopFault AND
   (ABS(backstopSignedSpeedRefMmps) >= machineConfig.backstopRunMinSpeedMmps) THEN

    // EN: The servo receives the signed speed reference directly.
    // PT: O servo recebe diretamente a referência de velocidade com sinal.
    backstopSpeedRefMmps := backstopSignedSpeedRefMmps;

    backstopRunFw :=
        backstopSignedSpeedRefMmps > 0.0;

    backstopRunRev :=
        backstopSignedSpeedRefMmps < 0.0;

ELSE

    backstopSpeedRefMmps := 0.0;

    backstopRunFw := FALSE;
    backstopRunRev := FALSE;

END_IF;

// EN: Enable the servo with the stacker system; drive-ready feedback is not used here
//     because it would create a circular enable dependency.
// PT: Habilita o servo com o sistema do stacker; o retorno de drive pronto não é usado
//     aqui porque criaria uma dependência circular de habilitação.
backstopDriveEnable := systemRunEnable AND safetyCircuitOk;


//==============================================================
// 13) Backstop plate lift solenoid
//==============================================================
// EN: Lift the backstop plate during backstop movement and homing.
//     Discharge conveyor protection can be ORed after all methods are called.
IF systemRunEnable AND
   (
       backstopRunFw OR
       backstopRunRev OR
       sheetStackDischargeConveyorRun OR
       (backstopControlState = 10) OR
       (backstopControlState = 11) OR
       (backstopControlState = 12) OR
       (backstopControlState = 13) OR
       (backstopControlState = 14)
   ) THEN

    backstopPlateUpSolenoid := TRUE;
    instTONBackstopDownDelay.IN := FALSE;

ELSE

    instTONBackstopDownDelay.IN := TRUE;

    IF instTONBackstopDownDelay.Q THEN

        backstopPlateUpSolenoid := FALSE;

    END_IF

END_IF;

instTONBackstopDownDelay(PT := T#200MS);
END_METHOD

//==============================================================
// COMPLEX STACKER — SPEED REFERENCE GENERATOR
// EN: Generates synchronized and sheet-stack separation speed references [m/min].
//==============================================================
METHOD _ConveyorSpeedControl
VAR
    rPackageComplete                  : BOOL;
    packageGapReady                   : BOOL;
    validCycleTimeS                   : REAL;

    sheetConveyorsSpeedUpReferenceMPM : REAL;

    sheetConveyor1BaseSpeedMPM        : REAL;
    sheetConveyor2BaseSpeedMPM        : REAL;
    sheetConveyor3BaseSpeedMPM        : REAL;
    sheetConveyor4BaseSpeedMPM        : REAL;
END_VAR


//==============================================================
// 1) Default event pulses
//==============================================================
sheetStackSeparationStarted         := FALSE;
sheetStackSeparationFinished        := FALSE;

sheetConveyor2SeparationStarted     := FALSE;
sheetConveyor2SeparationFinished    := FALSE;

sheetConveyor3SeparationStarted     := FALSE;
sheetConveyor3SeparationFinished    := FALSE;

sheetConveyor4SeparationStarted     := FALSE;
sheetConveyor4SeparationFinished    := FALSE;


//==============================================================
// 2) Edge detection
//==============================================================
rPackageComplete := packageCompleteCmd AND NOT packageCompleteCmdOld;
packageCompleteCmdOld := packageCompleteCmd;


//==============================================================
// 3) Enable and scan time
//==============================================================
speedControlEnabled :=
    sheetConveyor1Run AND
    sheetConveyor2Run AND
    sheetConveyor3Run AND
    sheetConveyor4Run AND
    safetyCircuitOk;

rampReset := NOT speedControlEnabled;


// EN: Read PLC scan time using OSCAT CYCLE_TIME.
instCycleTime(
    RST := resetCmd
);


// EN: Convert last cycle time from TIME/ms to seconds.
scanTimeMs := TIME_TO_REAL(instCycleTime.ct_last);

validCycleTimeS :=
    LIMIT(
        0.001,
        scanTimeMs / 1000.0,
        20.0
    );

scanTimeS := validCycleTimeS;


//==============================================================
// 4) Sheet length conversion
//==============================================================
// EN: Sheet length is kept converted for other calculations,
//     but it is no longer used as the separation tracking target.
sheetLengthM := MAX(0.0, sheetLengthMm) / 1000.0;


//==============================================================
// 5) Calculate normal stacker speed
//==============================================================
IF speedControlEnabled THEN

    normalStackerSpeedMPM :=
        LIMIT(
            machineConfig.minimumSpeedMPM,
            MAX(0.0, lineSpeedMPM) *
                MAX(0.0, machineConfig.stackerSpeedRatio),
            machineConfig.maximumSpeedMPM
        );

ELSE

    normalStackerSpeedMPM := 0.0;

END_IF;


//==============================================================
// 6) Calculate normal speed for each conveyor
//==============================================================
sheetConveyor1NormalSpeedMPM :=
    normalStackerSpeedMPM *
    MAX(0.0, machineConfig.sheetConveyor1SpeedTrim);

sheetConveyor2NormalSpeedMPM :=
    normalStackerSpeedMPM *
    MAX(0.0, machineConfig.sheetConveyor2SpeedTrim);

sheetConveyor3NormalSpeedMPM :=
    normalStackerSpeedMPM *
    MAX(0.0, machineConfig.sheetConveyor3SpeedTrim);

sheetConveyor4NormalSpeedMPM :=
    normalStackerSpeedMPM *
    MAX(0.0, machineConfig.sheetConveyor4SpeedTrim);


//==============================================================
// 6.1) Sheet conveyors speed-up reference
//==============================================================
// EN: Speed-up is added directly to conveyors 1/2/3 references.
//     It can work even when line speed is zero, as long as the
//     conveyor group is enabled.
IF speedControlEnabled AND sheetConveyorsSpeedUpCmd THEN

    sheetConveyorsSpeedUpReferenceMPM :=
        MAX(0.0, machineConfig.sheetConveyorsSpeedUpMPM);

ELSE

    sheetConveyorsSpeedUpReferenceMPM := 0.0;

END_IF;


//==============================================================
// 6.2) Base speed references including speed-up
//==============================================================
// EN: Base speed is the synchronized conveyor speed plus operator speed-up.
//     Separation tracking must use this base speed as reference.
sheetConveyor1BaseSpeedMPM :=
    sheetConveyor1NormalSpeedMPM + sheetConveyorsSpeedUpReferenceMPM;

sheetConveyor2BaseSpeedMPM :=
    sheetConveyor2NormalSpeedMPM + sheetConveyorsSpeedUpReferenceMPM;

sheetConveyor3BaseSpeedMPM :=
    sheetConveyor3NormalSpeedMPM + sheetConveyorsSpeedUpReferenceMPM;

sheetConveyor4BaseSpeedMPM :=
    sheetConveyor4NormalSpeedMPM + sheetConveyorsSpeedUpReferenceMPM;


//==============================================================
// 7) Calculate separation high speed
//==============================================================
// EN: Gap speed also receives the same speed-up reference.
//     This preserves the real gap differential while allowing operator boost.
sheetConveyor2GapSpeedMPM :=
    (sheetConveyor2NormalSpeedMPM * MAX(0.0, machineConfig.packageGapSpeedRatio)) +
    machineConfig.packageGapSpeedOffsetMPM +
    sheetConveyorsSpeedUpReferenceMPM;

sheetConveyor3GapSpeedMPM :=
    (sheetConveyor3NormalSpeedMPM * MAX(0.0, machineConfig.packageGapSpeedRatio)) +
    machineConfig.packageGapSpeedOffsetMPM +
    sheetConveyorsSpeedUpReferenceMPM;

sheetConveyor4GapSpeedMPM :=
    (sheetConveyor4NormalSpeedMPM * MAX(0.0, machineConfig.packageGapSpeedRatio)) +
    machineConfig.packageGapSpeedOffsetMPM +
    sheetConveyorsSpeedUpReferenceMPM;


//==============================================================
// 8) Calculate separation tracking target distances
//==============================================================
// EN: Separation tracking target is based on each conveyor length.
sheetConveyor2TargetDistanceM :=
    MAX(0.0, machineConfig.sheetConveyor2LengthM);

sheetConveyor3TargetDistanceM :=
    MAX(0.0, machineConfig.sheetConveyor3LengthM);

sheetConveyor4TargetDistanceM :=
    MAX(0.0, machineConfig.sheetConveyor4LengthM);


//==============================================================
// 9) Check separation ready conditions
//==============================================================
// EN: Compare gap speed against base speed, not normal speed.
//     Otherwise operator speed-up would be incorrectly counted as gap opening.
packageGapReady :=
    speedControlEnabled AND
    (sheetConveyor2TargetDistanceM > 0.0) AND
    (sheetConveyor3TargetDistanceM > 0.0) AND
    (sheetConveyor4TargetDistanceM > 0.0) AND
    ((sheetConveyor2GapSpeedMPM - sheetConveyor2BaseSpeedMPM) >= machineConfig.minimumOpeningSpeedMPM) AND
    ((sheetConveyor3GapSpeedMPM - sheetConveyor3BaseSpeedMPM) >= machineConfig.minimumOpeningSpeedMPM) AND
    ((sheetConveyor4GapSpeedMPM - sheetConveyor4BaseSpeedMPM) >= machineConfig.minimumOpeningSpeedMPM);

sheetStackSeparationReady := packageGapReady;


//==============================================================
// 10) Sheet stack separation state machine
//==============================================================
IF NOT speedControlEnabled THEN

    sheetStackSeparationState      := 'DISABLED';
    sheetStackSeparationStateCode  := -1;

    packageSeparationState         := 0;

    sheetStackSeparationActive     := FALSE;
    sheetStackBrakeActive          := FALSE;
    brakeValve                     := FALSE;

    sheetConveyor2SeparationActive := FALSE;
    sheetConveyor3SeparationActive := FALSE;
    sheetConveyor4SeparationActive := FALSE;

    sheetConveyor2HighSpeedActive  := FALSE;
    sheetConveyor3HighSpeedActive  := FALSE;
    sheetConveyor4HighSpeedActive  := FALSE;

    sheetConveyor2OpeningDistanceM := 0.0;
    sheetConveyor3OpeningDistanceM := 0.0;
    sheetConveyor4OpeningDistanceM := 0.0;

    sheetConveyor1TargetSpeedMPM   := 0.0;
    sheetConveyor2TargetSpeedMPM   := 0.0;
    sheetConveyor3TargetSpeedMPM   := 0.0;
    sheetConveyor4TargetSpeedMPM   := 0.0;


ELSE

    CASE packageSeparationState OF

        0: // NORMAL
            sheetStackSeparationState     := 'NORMAL';
            sheetStackSeparationStateCode := 0;

            sheetStackSeparationActive    := FALSE;
            sheetStackBrakeActive         := FALSE;
            brakeValve                    := FALSE;

            sheetConveyor2SeparationActive := FALSE;
            sheetConveyor3SeparationActive := FALSE;
            sheetConveyor4SeparationActive := FALSE;

            sheetConveyor2HighSpeedActive  := FALSE;
            sheetConveyor3HighSpeedActive  := FALSE;
            sheetConveyor4HighSpeedActive  := FALSE;

            sheetConveyor2OpeningDistanceM := 0.0;
            sheetConveyor3OpeningDistanceM := 0.0;
            sheetConveyor4OpeningDistanceM := 0.0;

            sheetConveyor1TargetSpeedMPM  := sheetConveyor1BaseSpeedMPM;
            sheetConveyor2TargetSpeedMPM  := sheetConveyor2BaseSpeedMPM;
            sheetConveyor3TargetSpeedMPM  := sheetConveyor3BaseSpeedMPM;
            sheetConveyor4TargetSpeedMPM  := sheetConveyor4BaseSpeedMPM;

            IF rPackageComplete AND packageGapReady THEN
                packageSeparationState := 10;
            END_IF


        10: // START_SHEET_STACK_SEPARATION
            sheetStackSeparationState     := 'START_SEPARATION';
            sheetStackSeparationStateCode := 10;

            sheetStackSeparationActive    := TRUE;
            sheetStackSeparationStarted   := TRUE;

            sheetStackBrakeActive         := TRUE;
            brakeValve                    := TRUE;

            // EN: Conveyor 2 tracking starts immediately.
            sheetConveyor2SeparationStarted := TRUE;

            sheetConveyor2SeparationActive  := TRUE;
            sheetConveyor3SeparationActive  := FALSE;
            sheetConveyor4SeparationActive  := FALSE;

            // EN: Conveyor 2 and 3 accelerate together from the beginning.
            sheetConveyor2HighSpeedActive   := TRUE;
            sheetConveyor3HighSpeedActive   := TRUE;
            sheetConveyor4HighSpeedActive   := TRUE;

            sheetConveyor2OpeningDistanceM  := 0.0;
            sheetConveyor3OpeningDistanceM  := 0.0;
            sheetConveyor4OpeningDistanceM  := 0.0;

            sheetConveyor1TargetSpeedMPM    := sheetConveyor1BaseSpeedMPM;
            sheetConveyor2TargetSpeedMPM    := sheetConveyor2GapSpeedMPM;
            sheetConveyor3TargetSpeedMPM    := sheetConveyor3GapSpeedMPM;
            sheetConveyor4TargetSpeedMPM    := sheetConveyor4GapSpeedMPM;

            packageSeparationState := 20;


        20: // SHEET_CONVEYOR_2_SEPARATION_TRACKING
            sheetStackSeparationState     := 'CONV2_TRACKING';
            sheetStackSeparationStateCode := 20;

            sheetStackSeparationActive    := TRUE;

            sheetStackBrakeActive         := TRUE;
            brakeValve                    := TRUE;

            sheetConveyor2SeparationActive := TRUE;
            sheetConveyor3SeparationActive := FALSE;
            sheetConveyor4SeparationActive := FALSE;

            sheetConveyor2HighSpeedActive  := TRUE;
            sheetConveyor3HighSpeedActive  := TRUE;
            sheetConveyor4HighSpeedActive  := TRUE;

            sheetConveyor1TargetSpeedMPM  := sheetConveyor1BaseSpeedMPM;
            sheetConveyor2TargetSpeedMPM  := sheetConveyor2GapSpeedMPM;
            sheetConveyor3TargetSpeedMPM  := sheetConveyor3GapSpeedMPM;
            sheetConveyor4TargetSpeedMPM  := sheetConveyor4GapSpeedMPM;

            IF sheetConveyor2OpeningDistanceM >= sheetConveyor2TargetDistanceM THEN

                // EN: Conveyor 2 tracking finished. Conveyor 2 returns to base speed.
                sheetConveyor2SeparationFinished := TRUE;

                sheetConveyor2SeparationActive   := FALSE;
                sheetConveyor2HighSpeedActive    := FALSE;

                sheetStackBrakeActive            := FALSE;
                brakeValve                       := FALSE;

                sheetConveyor2TargetSpeedMPM     := sheetConveyor2BaseSpeedMPM;

                // EN: Conveyor 3 tracking starts after conveyor 2 returns to sync.
                sheetConveyor3SeparationStarted := TRUE;
                sheetConveyor3OpeningDistanceM  := 0.0;

                packageSeparationState := 30;

            END_IF


        30: // SHEET_CONVEYOR_3_SEPARATION_TRACKING
            sheetStackSeparationState     := 'CONV3_TRACKING';
            sheetStackSeparationStateCode := 30;

            sheetStackSeparationActive    := TRUE;

            sheetStackBrakeActive         := FALSE;
            brakeValve                    := FALSE;

            sheetConveyor2SeparationActive := FALSE;
            sheetConveyor3SeparationActive := TRUE;
            sheetConveyor4SeparationActive := FALSE;

            sheetConveyor2HighSpeedActive  := FALSE;
            sheetConveyor3HighSpeedActive  := TRUE;
            sheetConveyor4HighSpeedActive  := TRUE;

            sheetConveyor1TargetSpeedMPM  := sheetConveyor1BaseSpeedMPM;
            sheetConveyor2TargetSpeedMPM  := sheetConveyor2BaseSpeedMPM;
            sheetConveyor3TargetSpeedMPM  := sheetConveyor3GapSpeedMPM;
            sheetConveyor4TargetSpeedMPM  := sheetConveyor4GapSpeedMPM;

            IF sheetConveyor3OpeningDistanceM >= sheetConveyor3TargetDistanceM THEN

                // EN: Conveyor 3 returns to base synchronized speed.
                sheetConveyor3TargetSpeedMPM := sheetConveyor3BaseSpeedMPM;

                // EN: Conveyor 4 tracking starts after conveyor 3 returns to sync.
                // PT: O rastreamento da esteira 4 inicia após a esteira 3 retornar ao sincronismo.
                sheetConveyor4SeparationStarted := TRUE;
                sheetConveyor4OpeningDistanceM := 0.0;

                packageSeparationState := 40;

            END_IF


        40: // SHEET_CONVEYOR_4_SEPARATION_TRACKING
            sheetStackSeparationState     := 'CONV4_TRACKING';
            sheetStackSeparationStateCode := 40;

            sheetStackSeparationActive    := TRUE;
            sheetStackBrakeActive         := FALSE;
            brakeValve                    := FALSE;

            sheetConveyor2SeparationActive := FALSE;
            sheetConveyor3SeparationActive := FALSE;
            sheetConveyor4SeparationActive := TRUE;

            sheetConveyor2HighSpeedActive := FALSE;
            sheetConveyor3HighSpeedActive := FALSE;
            sheetConveyor4HighSpeedActive := TRUE;

            sheetConveyor1TargetSpeedMPM := sheetConveyor1BaseSpeedMPM;
            sheetConveyor2TargetSpeedMPM := sheetConveyor2BaseSpeedMPM;
            sheetConveyor3TargetSpeedMPM := sheetConveyor3BaseSpeedMPM;
            sheetConveyor4TargetSpeedMPM := sheetConveyor4GapSpeedMPM;

            IF sheetConveyor4OpeningDistanceM >= sheetConveyor4TargetDistanceM THEN
                sheetConveyor4TargetSpeedMPM := sheetConveyor4BaseSpeedMPM;
                packageSeparationState := 50;
            END_IF


        50: // FINISH_SHEET_STACK_SEPARATION
            sheetStackSeparationState     := 'FINISH_SEPARATION';
            sheetStackSeparationStateCode := 50;

            sheetStackSeparationActive    := FALSE;
            sheetStackSeparationFinished  := TRUE;

            sheetStackBrakeActive         := FALSE;
            brakeValve                    := FALSE;

            sheetConveyor2SeparationActive  := FALSE;
            sheetConveyor3SeparationActive  := FALSE;
            sheetConveyor4SeparationActive  := FALSE;

            sheetConveyor2HighSpeedActive   := FALSE;
            sheetConveyor3HighSpeedActive   := FALSE;
            sheetConveyor4HighSpeedActive   := FALSE;

            sheetConveyor3SeparationFinished := TRUE;
            sheetConveyor4SeparationFinished := TRUE;

            sheetConveyor1TargetSpeedMPM  := sheetConveyor1BaseSpeedMPM;
            sheetConveyor2TargetSpeedMPM  := sheetConveyor2BaseSpeedMPM;
            sheetConveyor3TargetSpeedMPM  := sheetConveyor3BaseSpeedMPM;
            sheetConveyor4TargetSpeedMPM  := sheetConveyor4BaseSpeedMPM;

            packageSeparationState := 0;


    ELSE

        packageSeparationState := 0;

    END_CASE;

END_IF;


//==============================================================
// 11) Limit speed targets
//==============================================================
sheetConveyor1TargetSpeedMPM := LIMIT(
    machineConfig.minimumSpeedMPM,
    sheetConveyor1TargetSpeedMPM,
    machineConfig.maximumSpeedMPM
);

sheetConveyor2TargetSpeedMPM := LIMIT(
    machineConfig.minimumSpeedMPM,
    sheetConveyor2TargetSpeedMPM,
    machineConfig.maximumSpeedMPM
);

sheetConveyor3TargetSpeedMPM := LIMIT(
    machineConfig.minimumSpeedMPM,
    sheetConveyor3TargetSpeedMPM,
    machineConfig.maximumSpeedMPM
);

sheetConveyor4TargetSpeedMPM := LIMIT(
    machineConfig.minimumSpeedMPM,
    sheetConveyor4TargetSpeedMPM,
    machineConfig.maximumSpeedMPM
);


//==============================================================
// 12) Ramp sheet conveyor 1 speed reference
//==============================================================
instRampSheetConveyor1(
    X          := sheetConveyor1TargetSpeedMPM,
    A_UP       := MAX(0.0, machineConfig.rampAccelerationUpMPMps2),
    A_DN       := -MAX(0.0, machineConfig.rampAccelerationDownMPMps2),
    VU_MAX     := MAX(0.0, machineConfig.rampVelocityUpMaxMPMps),
    VD_MAX     := -MAX(0.0, machineConfig.rampVelocityDownMaxMPMps),
    LIMIT_HIGH := machineConfig.maximumSpeedMPM,
    LIMIT_LOW  := machineConfig.minimumSpeedMPM,
    RST        := rampReset,
    Y          => sheetConveyor1SpeedRefMPM
);


//==============================================================
// 13) Ramp sheet conveyor 2 speed reference
//==============================================================
instRampSheetConveyor2(
    X          := sheetConveyor2TargetSpeedMPM,
    A_UP       := MAX(0.0, machineConfig.rampAccelerationUpMPMps2),
    A_DN       := -MAX(0.0, machineConfig.rampAccelerationDownMPMps2),
    VU_MAX     := MAX(0.0, machineConfig.rampVelocityUpMaxMPMps),
    VD_MAX     := -MAX(0.0, machineConfig.rampVelocityDownMaxMPMps),
    LIMIT_HIGH := machineConfig.maximumSpeedMPM,
    LIMIT_LOW  := machineConfig.minimumSpeedMPM,
    RST        := rampReset,
    Y          => sheetConveyor2SpeedRefMPM
);


//==============================================================
// 14) Ramp sheet conveyor 3 speed reference
//==============================================================
instRampSheetConveyor3(
    X          := sheetConveyor3TargetSpeedMPM,
    A_UP       := MAX(0.0, machineConfig.rampAccelerationUpMPMps2),
    A_DN       := -MAX(0.0, machineConfig.rampAccelerationDownMPMps2),
    VU_MAX     := MAX(0.0, machineConfig.rampVelocityUpMaxMPMps),
    VD_MAX     := -MAX(0.0, machineConfig.rampVelocityDownMaxMPMps),
    LIMIT_HIGH := machineConfig.maximumSpeedMPM,
    LIMIT_LOW  := machineConfig.minimumSpeedMPM,
    RST        := rampReset,
    Y          => sheetConveyor3SpeedRefMPM
);


//==============================================================
// 15) Ramp sheet conveyor 4 speed reference
//==============================================================
instRampSheetConveyor4(
    X          := sheetConveyor4TargetSpeedMPM,
    A_UP       := MAX(0.0, machineConfig.rampAccelerationUpMPMps2),
    A_DN       := -MAX(0.0, machineConfig.rampAccelerationDownMPMps2),
    VU_MAX     := MAX(0.0, machineConfig.rampVelocityUpMaxMPMps),
    VD_MAX     := -MAX(0.0, machineConfig.rampVelocityDownMaxMPMps),
    LIMIT_HIGH := machineConfig.maximumSpeedMPM,
    LIMIT_LOW  := machineConfig.minimumSpeedMPM,
    RST        := rampReset,
    Y          => sheetConveyor4SpeedRefMPM
);


//==============================================================
// 16) Calculate real separation tracking speed using ramped references
//==============================================================
// EN: Only the real speed differential above the base speed moves the
//     separation point through the conveyors.
//     Operator speed-up is already included in base speed, so it is not
//     counted as gap opening.
sheetConveyor2OpeningSpeedMPM :=
    MAX(0.0, sheetConveyor2SpeedRefMPM - sheetConveyor2BaseSpeedMPM);

sheetConveyor3OpeningSpeedMPM :=
    MAX(0.0, sheetConveyor3SpeedRefMPM - sheetConveyor3BaseSpeedMPM);

sheetConveyor4OpeningSpeedMPM :=
    MAX(0.0, sheetConveyor4SpeedRefMPM - sheetConveyor4BaseSpeedMPM);


//==============================================================
// 17) Integrate real separation tracking distance
//==============================================================
IF speedControlEnabled THEN

    IF packageSeparationState = 20 THEN

        IF sheetConveyor2OpeningSpeedMPM >= machineConfig.minimumOpeningSpeedMPM THEN

            sheetConveyor2OpeningDistanceM :=
                sheetConveyor2OpeningDistanceM +
                (sheetConveyor2OpeningSpeedMPM / 60.0) * scanTimeS;

        END_IF

    ELSIF packageSeparationState = 30 THEN

        IF sheetConveyor3OpeningSpeedMPM >= machineConfig.minimumOpeningSpeedMPM THEN

            sheetConveyor3OpeningDistanceM :=
                sheetConveyor3OpeningDistanceM +
                (sheetConveyor3OpeningSpeedMPM / 60.0) * scanTimeS;

        END_IF

    ELSIF packageSeparationState = 40 THEN

        IF sheetConveyor4OpeningSpeedMPM >= machineConfig.minimumOpeningSpeedMPM THEN

            sheetConveyor4OpeningDistanceM :=
                sheetConveyor4OpeningDistanceM +
                (sheetConveyor4OpeningSpeedMPM / 60.0) * scanTimeS;

        END_IF

    END_IF

END_IF;


//==============================================================
// 18) Publish tracking distances to outputs
//==============================================================
sheetConveyor2TrackingDistanceM := sheetConveyor2OpeningDistanceM;
sheetConveyor3TrackingDistanceM := sheetConveyor3OpeningDistanceM;
sheetConveyor4TrackingDistanceM := sheetConveyor4OpeningDistanceM;
END_METHOD

//==============================================================
// COMPLEX STACKER - ELEVATOR CONTROL
// EN: Controls homing, manual movement, automatic leveling,
//     discharge positioning and magnetic brake timing.
// PT: Controla homing, movimento manual, nivelamento automático,
//     posicionamento de descarga e temporização do freio magnético.
//
// Signed speed: positive = up; negative = down.
// Velocidade com sinal: positivo = subir; negativo = descer.
//
// State code:
// 0  = STOP
// 10 = HOME_DOWN_SEARCH
// 11 = HOME_RELEASE_SENSOR
// 12 = HOME_SETTLE
// 13 = HOME_SET_ENCODER
// 14 = HOME_MOVE_TO_UPPER_POSITION
// 20 = MANUAL
// 30 = AUTO_LEVELING
// 40 = DISCHARGE_POSITIONING
// 90 = FAULT
//==============================================================
METHOD _ElevatorControl
//==============================================================
// 1) Default internal commands
//==============================================================
elevatorSignedSpeedRefMmps := 0.0;
elevatorSetEncoderPositionTrigger := FALSE;
elevatorManualLowSpeedZoneActive := FALSE;


//==============================================================
// 2) Homing request and lower sensor edge detection
//==============================================================
elevatorHomeRequestCombined :=
    systemRunEnable AND
    (
        elevatorHomeCmd OR
        (
            elevatorAutoCmd AND
            elevatorAutoHomeRequest
        )
    );

rElevatorHome :=
    elevatorHomeRequestCombined AND
    NOT elevatorHomeRequestCombinedOld;

elevatorHomeRequestCombinedOld := elevatorHomeRequestCombined;

elevatorHomeLimitReached := elevatorLowerLimit;

elevatorHomeLimitFallingEdge :=
    elevatorHomeLimitOld AND
    NOT elevatorHomeLimitReached;

elevatorHomeLimitOld := elevatorHomeLimitReached;


//==============================================================
// 2.1) Manual command rearm
//==============================================================
// EN: Manual commands held during homing or active discharge positioning
//     must be released before a new manual movement can start.
//     Waiting for stack separation keeps leveling and manual control active.
// PT: Comandos manuais mantidos durante homing ou posicionamento ativo de
//     descarte devem ser liberados antes que um novo movimento manual inicie.
//     A espera pela separação mantém o nivelamento e o controle manual ativos.
IF NOT systemRunEnable OR
   NOT safetyCircuitOk OR
   NOT elevatorDriveOk OR
   elevatorFault OR
   (
        (elevatorControlState >= 10) AND
        (elevatorControlState <= 14)
   ) OR
   (elevatorControlState = 40) OR
   (elevatorControlState = 90) OR
   elevatorTargetOverrideActive OR
   sheetStackDischargeActive THEN

    elevatorManualCommandArmed := FALSE;

ELSIF NOT elevatorUpCmd AND
      NOT elevatorDownCmd THEN

    elevatorManualCommandArmed := TRUE;

END_IF;

elevatorManualCommandRequest :=
    elevatorManualCommandArmed AND
    (elevatorUpCmd OR elevatorDownCmd);


//==============================================================
// 3) Movement permissions
//==============================================================
elevatorUpAllowed :=
    systemRunEnable AND
    safetyCircuitOk AND
    elevatorDriveOk AND
    NOT elevatorUpperLimit AND
    NOT elevatorUpperSafetyLimit AND
    NOT backstopMaterialInterlockSensor AND
    (
        (NOT elevatorHomed) OR
        (elevatorPositionMm < machineConfig.elevatorMaxPositionMm)
    );

elevatorDownAllowed :=
    systemRunEnable AND
    safetyCircuitOk AND
    elevatorDriveOk AND
    NOT elevatorLowerLimit AND
    NOT elevatorLowerSafetyLimit AND
    (
        (NOT elevatorHomed) OR
        (elevatorPositionMm > machineConfig.elevatorMinPositionMm)
    );

// EN: Homing search ignores the normal lower limit until it is detected.
// PT: A busca de home ignora o limite inferior normal até detectá-lo.
elevatorHomeDownAllowed :=
    systemRunEnable AND
    safetyCircuitOk AND
    elevatorDriveOk AND
    NOT elevatorLowerSafetyLimit;

// EN: Upward release respects the backstop material interlock.
// PT: A liberação para cima respeita o intertravamento de material do backstop.
elevatorHomeReleaseAllowed :=
    systemRunEnable AND
    safetyCircuitOk AND
    elevatorDriveOk AND
    NOT elevatorUpperLimit AND
    NOT elevatorUpperSafetyLimit AND
    NOT backstopMaterialInterlockSensor;

//==============================================================
// 4) Target and position feedback
//==============================================================
IF elevatorControlState = 14 THEN

    elevatorTargetPositionMm := machineConfig.elevatorMaxPositionMm;

ELSIF elevatorTargetOverrideActive THEN

    elevatorTargetPositionMm :=
        LIMIT(
            machineConfig.elevatorMinPositionMm,
            elevatorTargetOverridePositionMm,
            machineConfig.elevatorMaxPositionMm
        );

ELSE

    elevatorTargetPositionMm :=
        LIMIT(
            machineConfig.elevatorMinPositionMm,
            elevatorPositionMm,
            machineConfig.elevatorMaxPositionMm
        );

END_IF;

elevatorPositionErrorMm :=
    elevatorTargetPositionMm - elevatorPositionMm;

elevatorAbsPositionErrorMm := ABS(elevatorPositionErrorMm);

// EN: Proportional position control with independent directional limits.
//     No minimum speed is forced; the servo may receive zero near the target.
// PT: Controle proporcional de posição com limites independentes por sentido.
//     Não força velocidade mínima; o servo pode receber zero próximo ao alvo.
elevatorRawSpeedRefMmps :=
    elevatorPositionErrorMm * MAX(0.0, machineConfig.elevatorPositionKp);

elevatorRawSpeedRefMmps :=
    LIMIT(
        -ABS(machineConfig.elevatorAutomaticDownSpeedMmps),
        elevatorRawSpeedRefMmps,
        ABS(machineConfig.elevatorAutomaticUpSpeedMmps)
    );

